TYPE TIMER_EVENT :
STRUCT
	TYP : BYTE;
	CHANNEL : BYTE;
	DAY : BYTE;
	START : TOD;
	DURATION : TIME;
	LAND : BYTE;
	LOR : BYTE;
	LAST : DT;
END_STRUCT
END_TYPE

(* stored: Version 1.1.0.1
   DUT TIMER_EVENT: Id {f38f251c-6548-4f5c-b694-00cf4a86bda4} *)
